// TwinCAT 3 PLC project Internship
// ProgramVersion: 3.1.4024.0
// libraries:
//   Tc2_Standard, * (Beckhoff Automation GmbH)
//   Tc2_System, * (Beckhoff Automation GmbH)
//   Tc3_Module, * (Beckhoff Automation GmbH)
// project tree:
//   Control/ FB_ControlSignal.TcPOU, FB_FeedForward.TcPOU, FB_PID.TcPOU, FB_Running.TcPOU (not stored), G_Mode.TcGVL
//   Filtering/ FB_Filtering.TcPOU, G_Filtered.TcGVL
//   GVL/ E_Mode.TcDUT, G_Enables.TcGVL, G_FilterConstants.TcGVL, G_OPC.TcGVL, G_Parameter.TcGVL
//   Inputs/Function Blocks/ FB_JoystickInputScaling.TcPOU, FB_Normalize.TcPOU, FB_Normalize_Joystick.TcPOU, FB_PositionInputScaling.TcPOU
//   Inputs/ G_Inputs.TcGVL
//   MotionRef/ FB_AutoClock.TcPOU, FB_DeadbandTester.TcPOU, FB_InitialPos.TcPOU, FB_MotionRef.TcPOU, FB_RunClock.TcPOU
//   Outputs/ FB_ValveOutput.TcPOU, G_Output.TcGVL
//   / PlcTask.TcTTO
//   Programs/ MAIN.TcPOU, P_ControlBlock.TcPOU, P_FeedForward.TcPOU, P_Filtering.TcPOU, P_Inputs.TcPOU, P_Modes.TcPOU, P_Output.TcPOU, P_PID.TcPOU, P_RunClock.TcPOU
//   XML/ FB_Derivator.TcPOU, G_Init.TcGVL, FB_Integrator.TcPOU
// real-time tasks:
//   TASK PlcTask: cycle T#1ms, priority 20, ADS port 350
// I/O:
//   DEVICE Device 3 (EtherCAT), AmsNetId 192.168.1.1.4.1
//     RIO (EK1100) [EK1100 EtherCAT Coupler (2A E-Bus)]
//       DI (EL1008) [EL1008 8Ch. Dig. Input 24V, 3ms]
//       DO (EL2008) [EL2008 8Ch. Dig. Output 24V, 0.5A]
//       AI1 (EL3068) [EL3068 8Ch. Ana. Input 0-10V]
//       AI2 (EL3068) [EL3068 8Ch. Ana. Input 0-10V]
//       AI3 (EL3174) [EL3174 4Ch. Ana. Input +/-10V Diff., +/-20mA SingleEnded, 16 Bit]
//       AO (EL4104) [EL4104 4Ch. Ana. Output 0-10V, 16bit]
//       End Cap (EL9011) [EL9011 End Terminal]
// variable links:
//   Internship/Internship Instance <-> Device 3 (EtherCAT)/RIO (EK1100)/AI1 (EL3068)
//     PlcTask Inputs/G_Inputs.nRawJoystick <-> AI Standard Channel 2/Value
//     PlcTask Inputs/G_Inputs.nRawPistonPosition <-> AI Standard Channel 3/Value
//   Internship/Internship Instance <-> Device 3 (EtherCAT)/RIO (EK1100)/AI2 (EL3068)
//     PlcTask Inputs/G_Inputs.nRawPa <-> AI Standard Channel 4/Value
//     PlcTask Inputs/G_Inputs.nRawPaLower <-> AI Standard Channel 5/Value
//     PlcTask Inputs/G_Inputs.nRawPb <-> AI Standard Channel 6/Value
//     PlcTask Inputs/G_Inputs.nRawPs <-> AI Standard Channel 1/Value
//   Internship/Internship Instance <-> Device 3 (EtherCAT)/RIO (EK1100)/AO (EL4104)
//     PlcTask Outputs/G_Output.nValveOutput <-> AO Output Channel 1/Analog output
//   Internship/Internship Instance <-> Device 3 (EtherCAT)/RIO (EK1100)/DI (EL1008)
//     PlcTask Inputs/G_Inputs.bAuto <-> Channel 1/Input
//     PlcTask Inputs/G_Inputs.bManual <-> Channel 2/Input
//     PlcTask Inputs/G_Inputs.bStartButton <-> Channel 3/Input
//     PlcTask Inputs/G_Inputs.bStopButton <-> Channel 4/Input
//   Internship/Internship Instance <-> Device 3 (EtherCAT)/RIO (EK1100)/DO (EL2008)
//     PlcTask Outputs/G_Output.bGreenLight <-> Channel 1/Output
//     PlcTask Outputs/G_Output.bRedLight <-> Channel 2/Output
//     PlcTask Outputs/G_Output.bRunning <-> Channel 3/Output

CONFIGURATION Internship
    RESOURCE PLC ON TwinCAT3
        TASK PlcTask(INTERVAL := T#1ms, PRIORITY := 20);
        PROGRAM MAIN WITH PlcTask : MAIN;
    END_RESOURCE
END_CONFIGURATION

// ---- GVL/E_Mode.TcDUT
{attribute 'qualified_only'}
{attribute 'strict'}
TYPE E_Mode :
(
	Off := 0,
	Auto := 1,
	Manuel := 2
);
END_TYPE

// ---- Control/G_Mode.TcGVL
{attribute 'qualified_only'}
VAR_GLOBAL
	bRunning : BOOL;
	bManual : BOOL;
	bAuto : BOOL;
END_VAR

// ---- Filtering/G_Filtered.TcGVL
{attribute 'qualified_only'}
VAR_GLOBAL
	fPressureSupplyFiltered		: LREAL;
	fPressurePistonSideFiltered : LREAL;
	fPressureRodSideFiltered 	: LREAL;
	fValveOutputFiltered		: LREAL;
	fValveOutputUnfiltered		: LREAL;
END_VAR

// ---- GVL/G_Enables.TcGVL
{attribute 'qualified_only'}
VAR_GLOBAL
	// Enables
	bEnablePID 		: BOOL := FALSE; // Enable PID Control
	bEnableU 		: BOOL := FALSE; // Enable Signal to Valve
	bEnableFF 		: BOOL := FALSE; // Enable FeedForward
	bMotionSelect 	: BOOL := FALSE; // Switch Motion Reference generator
	bEnableComp 	: BOOL := FALSE; // Driving with Compensator
	bDeadBand 		: BOOL := FALSE; // Enable Dead Band Testing
END_VAR

// ---- GVL/G_FilterConstants.TcGVL
{attribute 'qualified_only'}
VAR_GLOBAL
	// Filter constants
	fPressureFilterNum :LREAL := 0.003137;
	fPressureFilterDenz : LREAL := 1.0;
	fPressureFilterDen : LREAL := -0.9969;
	fPressureFilterInit : LREAL := 0.0;
	
	fSignalFilterNum : LREAL := 0.09516;
	fSignalFilterDenz : LREAL := 1.0;
	fSignalFilterDen : LREAL := -0.9048;
	fSignalFilterInit : LREAL := 0.0;
	
	fDerivatorFilterNum : LREAL := 0.0009995;
	fDerivatorFilterDenz : LREAL := 1.0;
	fDerivatorFilterDen : LREAL := -0.999;
	fDerivatorFilterInit : LREAL := 0.0;	
END_VAR

// ---- GVL/G_OPC.TcGVL
{attribute 'qualified_only'}
VAR_GLOBAL
	
	// Unfiltered Pressures
	fPa : LREAL;
	fPb : LREAL;
	fPs : LREAL;
	fPaLower : LREAL;
	
	// Filtered Pressures
	fPaFiltered : LREAL;
	fPbFiltered : LREAL;
	fPsFiltered : LREAL;
	fPaLowerFiltered : LREAL;
	
	
	fPistonPosition : LREAL;
	fJoystick : LREAL;
	
	fXRef : LREAL;
	fXDotRef : LREAL;
	
	fU : LREAL;
	fTime : LREAL;
	fError : LREAL;
	fSignalPID : LREAL;
	fUFF : LREAL;
END_VAR

// ---- GVL/G_Parameter.TcGVL
{attribute 'qualified_only'}
VAR_GLOBAL
	// Motion Ref
	fAmplitude : LREAL := 0.1;
	fMean : LREAL := 0.2;
	fFrequency : LREAL := 0.05;
	
	
	// Valve Values
	fQMaxDown : LREAL := 15.9;
	fQMaxUp : LREAL := 24.4;
	fDeadUp : LREAL := 0.13;
	fDeadDown : LREAL := 0.13;
	
	fMaxSpeed : LREAL := 0.01; // [m/s] 
	
	// Deadband test
	fConst : LREAL := 0.0; // [-1, 1]

	
	fCycleTime : LREAL := 0.001; // Time Step [s]
	fQConst : LREAL := 15;
	
	// PID-constants
	Kp : LREAL := 14.0; 	// P
	Ki : LREAL := 0.0;		// I
	Kd : LREAL := 0.0;		// D
	
	
	
	
END_VAR

// ---- Inputs/G_Inputs.TcGVL
{attribute 'qualified_only'}
VAR_GLOBAL
	// Mode Selector
	bManual 			AT %I* : BOOL;
	bAuto	 			AT %I* : BOOL;
	bStartButton		AT %I* : BOOL;
	bStopButton			AT %I* : BOOL;
	
	// Raw Pressure Values
	nRawPa 				AT %I*	: INT;
	nRawPb				AT %I*	: INT;
	nRawPs				AT %I*	: INT;
	nRawPaLower				AT %I* 	: INT;
	
	// Raw Position Values
	nRawPistonPosition 	AT %I*	: INT;
	nRawJoystick		AT %I*	: INT;
END_VAR

// ---- Outputs/G_Output.TcGVL
{attribute 'qualified_only'}
VAR_GLOBAL
	// Digital Outputs
	bGreenLight 			AT %Q* : BOOL;
	bRedLight 				AT %Q* : BOOL;
	
	// Analog Outputs
	nValveOutput 			AT %Q* : INT; 
	bRunning				AT %Q* : BOOL;
END_VAR

// ---- XML/G_Init.TcGVL
VAR_GLOBAL CONSTANT
	SS_INITIALIZE: SINT := 0;
	SS_STEP: SINT := 1;
END_VAR

// ---- Programs/MAIN.TcPOU
PROGRAM MAIN
VAR
END_VAR

P_Inputs();
P_Filtering();
P_ControlBlock();
P_Output();
//P_RunClock();
P_Modes();
P_PID();
P_FeedForward();

END_PROGRAM

// ---- Programs/P_Inputs.TcPOU
PROGRAM P_Inputs
VAR
	fbNormPa :  FB_Normalize;
	fbNormPb :  FB_Normalize;
	fbNormPs :  FB_Normalize;
	
	fbNormPistonPosition : FB_PositionInputScaling;
	fbJoystick : FB_JoystickInputScaling;

	fPa : LREAL;
	fPb : LREAL;
	fPs : LREAL;
	
	fPistonPosition : LREAL;
END_VAR

fbNormPa(
	nRawInput := G_Inputs.nRawPa,
	fMaxValue := 400.0, 			// [Bar]
	fNormalizedInput => G_OPC.fPa
);

fbNormPb(
	nRawInput := G_Inputs.nRawPb,
	fMaxValue := 400.0, 			// [Bar]
	fNormalizedInput => G_OPC.fPb
);

fbNormPs(
	nRawInput := G_Inputs.nRawPs,
	fMaxValue := 400.0, 			// [Bar]
	fNormalizedInput => G_OPC.fPs
);

fbNormPistonPosition(
	nRawInput := G_Inputs.nRawPistonPosition,
	fOutput => G_OPC.fPistonPosition
);
	
fbJoystick(
	nRawInput := G_Inputs.nRawJoystick,
	bEnable := G_Inputs.bManual,
	fOutput => G_OPC.fJoystick
);

END_PROGRAM

// ---- Inputs/Function Blocks/FB_Normalize.TcPOU
FUNCTION_BLOCK FB_Normalize
VAR_INPUT
	nRawInput : INT;
	fMaxValue : LREAL;
END_VAR
VAR_OUTPUT
	fNormalizedInput : LREAL;
END_VAR
VAR
END_VAR

fNormalizedInput := (fMaxValue	* INT_TO_LREAL(nRawInput)) / 32767.0;

fNormalizedInput := LIMIT(0, fNormalizedInput, fMaxValue);

END_FUNCTION_BLOCK

// ---- Inputs/Function Blocks/FB_PositionInputScaling.TcPOU
FUNCTION_BLOCK FB_PositionInputScaling
VAR_INPUT
	nRawInput : INT;
END_VAR
VAR_OUTPUT
	fOutput : LREAL;
END_VAR
VAR
	fRawInput : LREAL;
	fNormalizedInput: LREAL;
	fMaxInputValue 			: LREAL := 16099.0;
	fMinInputValue			: LREAL := 125.0;
	fMaxOutputValue  		: LREAL := 0.5;
	fMinOutputValue  		: LREAL := 0.0;		
END_VAR

fRawInput := INT_TO_LREAL(nRawInput);

fNormalizedInput := (fRawInput - fMinInputValue) / (fMaxInputValue - fMinInputValue);

fOutput := LIMIT(fMinOutputValue, fMinOutputValue + fNormalizedInput*(fMaxOutputValue - fMinOutputValue), fMaxOutputValue);

END_FUNCTION_BLOCK

// ---- Inputs/Function Blocks/FB_JoystickInputScaling.TcPOU
FUNCTION_BLOCK FB_JoystickInputScaling
VAR_INPUT
	bEnable : BOOL;
	nRawInput : INT;
END_VAR
VAR_OUTPUT
	fOutput : LREAL;
END_VAR
VAR
	fRawInput : LREAL;
	fTempInput : LREAL;
	fTempOutput : LREAL;
	fMaxInputValue			: LREAL := 14746.0;
	fMinInputValue 			: LREAL := 1617.0;
	fNeutralInputValue  	: LREAL := 8160.0;
	fNeutralDeadband		: LREAL := 100.0;
	fMaxOutputValue  		: LREAL := 1.0;
	fMinOutputValue  		: LREAL := -1.0;
	fNeutralOutputValue  	: LREAL := 0.0;
END_VAR

fRawInput := INT_TO_LREAL(nRawInput);

fTempInput := fRawInput - fNeutralInputValue;

IF fTempInput > fNeutralDeadband THEN
	fTempOutput := fTempInput/(fMaxInputValue - fNeutralInputValue);
ELSIF fTempInput < -fNeutralDeadband THEN	
	fTempOutput := fTempInput/(fNeutralInputValue - fMinInputValue);
ELSE
	fTempOutput := 0.0;
END_IF

IF NOT(bEnable) THEN
	fOutput := 0.0;
ELSE
	fOutput := LIMIT(fMinOutputValue, fTempOutput, fMaxOutputValue);
END_IF

END_FUNCTION_BLOCK

// ---- Programs/P_Filtering.TcPOU
PROGRAM P_Filtering
VAR
	//fbControlBlock : c_FB_ControlBlockWithMonito;
	fbFilterPa : FB_Filtering;
	fbFilterPb : FB_Filtering;
	fbFilterPs : FB_Filtering;
	fbFilterU : FB_Filtering;
	fbFilterPaLower : FB_Filtering;
END_VAR

fbFilterPa(
	ssMethodType := 1,
	Signal := G_OPC.fPa,
	Num := G_FilterConstants.fPressureFilterNum,
	Denz := G_FilterConstants.fPressureFilterDenz,
	Den := G_FilterConstants.fPressureFilterDen,
	Initial := G_FilterConstants.fPressureFilterInit,
	
	Signal_Filtered => G_Filtered.fPressurePistonSideFiltered,
	Signal_Filtered => G_OPC.fPaFiltered
);

fbFilterPb(
	ssMethodType := 1,
	Signal := G_OPC.fPb,
	Num := G_FilterConstants.fPressureFilterNum,
	Denz := G_FilterConstants.fPressureFilterDenz,
	Den := G_FilterConstants.fPressureFilterDen,
	Initial := G_FilterConstants.fPressureFilterInit,
	
	Signal_Filtered => G_Filtered.fPressureRodSideFiltered,
	Signal_Filtered => G_OPC.fPbFiltered
);

fbFilterPs(
	ssMethodType := 1,
	Signal := G_OPC.fPs,
	Num := G_FilterConstants.fPressureFilterNum,
	Denz := G_FilterConstants.fPressureFilterDenz,
	Den := G_FilterConstants.fPressureFilterDen,
	Initial := G_FilterConstants.fPressureFilterInit,
	
	Signal_Filtered => G_Filtered.fPressureSupplyFiltered,
	Signal_Filtered => G_OPC.fPsFiltered
);

fbFilterPaLower(
	ssMethodType := 1,
	Signal := G_OPC.fPaLower,
	Num := G_FilterConstants.fPressureFilterNum,
	Denz := G_FilterConstants.fPressureFilterDenz,
	Den := G_FilterConstants.fPressureFilterDen,
	Initial := G_FilterConstants.fPressureFilterInit,
	
	Signal_Filtered => G_Filtered.fPressureSupplyFiltered,
	Signal_Filtered => G_OPC.fPaLowerFiltered
);

//fbFilterU(
//	ssMethodType := 1,
//	Signal := G_Filtered.fValveOutputUnfiltered,
//	Num := G_FilterConstants.fSignalFilterNum,
//	Denz := G_FilterConstants.fSignalFilterDenz,
//	Den := G_FilterConstants.fSignalFilterDen,
//	Initial := G_FilterConstants.fSignalFilterInit,
//	
//	Signal_Filtered => G_Filtered.fValveOutputFiltered,
//	Signal_Filtered => G_OPC_UA.fFilteredSignal
//);

END_PROGRAM

// ---- Filtering/FB_Filtering.TcPOU
FUNCTION_BLOCK FB_Filtering
VAR_INPUT
	ssMethodType: SINT;
	Signal: LREAL;
	Num: LREAL;
	DenZ: LREAL;
	Den: LREAL;
	Initial: LREAL;
END_VAR
VAR_OUTPUT
	Signal_Unfiltered: LREAL;
	Signal_Filtered: LREAL;
END_VAR
VAR
	DiscreteTransferFcn1_icLoad: USINT;
	DiscreteTransferFcn1_states: LREAL;
	c_TmpSignalConversionAtDisc: ARRAY[0..1] OF LREAL;
END_VAR



CASE ssMethodType OF
    SS_INITIALIZE: 
        (* SystemInitialize for Atomic SubSystem: '<Root>/FB_Filtering' *)
        (* InitializeConditions for DiscreteTransferFcn: '<S1>/Discrete Transfer Fcn1' *)
        DiscreteTransferFcn1_icLoad := 1;
        (* End of SystemInitialize for SubSystem: '<Root>/FB_Filtering' *)
    SS_STEP: 
        (* Outputs for Atomic SubSystem: '<Root>/FB_Filtering' *)
        (* SignalConversion: '<S1>/TmpSignal ConversionAtDiscrete Transfer Fcn1Inport3' *)
        c_TmpSignalConversionAtDisc[0] := DenZ;
        c_TmpSignalConversionAtDisc[1] := Den;
        (* DiscreteTransferFcn: '<S1>/Discrete Transfer Fcn1' *)

        IF DiscreteTransferFcn1_icLoad <> 0 THEN 
            DiscreteTransferFcn1_states := Initial;
        END_IF;

        Signal_Filtered := Num * DiscreteTransferFcn1_states;
        (* End of DiscreteTransferFcn: '<S1>/Discrete Transfer Fcn1' *)
        

        (* SignalConversion: '<S1>/Signal' incorporates:
         *  Outport: '<Root>/Signal_Unfiltered' *)
        Signal_Unfiltered := Signal;
        (* Update for DiscreteTransferFcn: '<S1>/Discrete Transfer Fcn1' incorporates:
         *  SignalConversion: '<S1>/Signal' *)
        DiscreteTransferFcn1_icLoad := 0;
        DiscreteTransferFcn1_states := Signal - (c_TmpSignalConversionAtDisc[1] * DiscreteTransferFcn1_states);
        (* End of Outputs for SubSystem: '<Root>/FB_Filtering' *)
END_CASE;

END_FUNCTION_BLOCK

// ---- Programs/P_ControlBlock.TcPOU
PROGRAM P_ControlBlock
VAR
	fbDeadBandTester : FB_DeadbandTester;
	fbAutoClock : FB_AutoClock;
	fbMotionRef : FB_MotionRef;
	fbControl : FB_ControlSignal;
	fbInitialPos : FB_InitialPos;
END_VAR


fbControl(
	bEnableU := G_Enables.bEnableU,
	fQMaxUp := G_Parameter.fQMaxUp,
	fQMaxDown := G_Parameter.fQMaxDown,
	fDeadUp := G_Parameter.fDeadUp,
	fDeadDown := G_Parameter.fDeadDown,
);


IF G_Mode.bAuto AND G_Mode.bRunning THEN

fbInitialPos(
	bEnable := G_Inputs.bStartButton,
	fCurrentPos := G_OPC.fPistonPosition
);

fbAutoClock(
	fStart := G_Inputs.bStartButton,
	fRunning := G_Mode.bRunning,
	fCycle := G_Parameter.fCycleTime
);

fbMotionRef(
	fTime := fbAutoClock.fTime,
	fAmplitude := G_Parameter.fAmplitude,
	fInitialPos := fbInitialPos.fInitialPos,
	fFrequency := G_Parameter.fFrequency,
	fXDotRef => G_OPC.fXDotRef,
	fXRef => G_OPC.fXRef 
);

fbControl(
	fUFF := G_OPC.fUFF,
	fPID := G_OPC.fSignalPID,
	
	fU => G_OPC.fU
);

ELSIF G_Mode.bManual AND G_Mode.bRunning THEN

fbInitialPos(
	bEnable := G_Inputs.bStartButton,
	fCurrentPos := G_OPC.fPistonPosition
);

fbDeadBandTester(
	fInput := G_OPC.fJoystick,
	bEnable := G_Enables.bDeadBandTest,
	fConst := G_Parameter.fConst,
	fOutput => G_OPC.fU
);

//fbControl(
//	fUFF := G_OPC.fJoystick * G_Parameter.fMaxSpeed,
//	fPID := G_OPC.fSignalPID,
	
//	fU => G_OPC.fU
//);


END_IF

END_PROGRAM

// ---- MotionRef/FB_DeadbandTester.TcPOU
FUNCTION_BLOCK FB_DeadbandTester
VAR_INPUT
	fInput : LREAL;
	bEnable : BOOL;
	fConst : LREAL;
END_VAR
VAR_OUTPUT
	fOutput : LREAL;
END_VAR
VAR
	
END_VAR

IF bEnable THEN
	fOutput := fInput;
ELSE
	fOutput := fConst;
END_IF

END_FUNCTION_BLOCK

// ---- MotionRef/FB_AutoClock.TcPOU
FUNCTION_BLOCK FB_AutoClock
VAR_INPUT
	fStart : BOOL;
	fRunning : BOOL;
	fCycle : LREAL;
END_VAR
VAR_OUTPUT
	fTime : LREAL;
END_VAR
VAR
END_VAR


IF NOT(fStart) OR NOT(fRunning) THEN
	fTime := 0.0;
ELSIF fStart AND fRunning THEN
	fTime := fTime + fCycle;		
END_IF

END_FUNCTION_BLOCK

// ---- MotionRef/FB_MotionRef.TcPOU
FUNCTION_BLOCK FB_MotionRef
VAR_INPUT
	fTime : LREAL;
	fAmplitude : LREAL;
	fFrequency : LREAL;
	fInitialPos : LREAL;
END_VAR
VAR_OUTPUT
	fXDotRef : LREAL;
	fXRef : LREAL;
END_VAR
VAR
	fPI : LREAL := 3.1415;
	fMean : LREAL;
END_VAR

fMean := fAmplitude + fInitialPos; 
fXRef := fMean - fAmplitude * COS(2*fPI * fFrequency * fTime);
fXDotRef := 2 * fPI *fFrequency * fAmplitude * SIN(2*fPI * fFrequency * fTime);

END_FUNCTION_BLOCK

// ---- Control/FB_ControlSignal.TcPOU
FUNCTION_BLOCK FB_ControlSignal
VAR_INPUT
	fUFF : LREAL;
	fPID : LREAL;
	bEnableU : BOOL;
	fQMaxUp 	: LREAL; // Needs to be positive (22)
	fQMaxDown 	: LREAL; // Needs to be positive (15)
	fDeadUp		: LREAL; // Needs to be positive (0.155)
	fDeadDown 	: LREAL; // Needs to be positive (0.18)
END_VAR
VAR_OUTPUT
	fU : LREAL;
END_VAR
VAR

	fUTemp : LREAL;
	fUTemp2 : LREAL;
	fUMax : LREAL := 0.9;
END_VAR

IF bEnableU THEN
	fUTemp := fUFF - fPID;
	
	// Deadband compensation
	IF fUTemp < 0.0 THEN	// Upwards
		fUTemp2 := fUTemp - fDeadUp;
	ELSIF fUTemp > 0.0 THEN // Downwards
		fUTemp2 := fUTemp + fDeadDown;
	ELSE
		fUTemp2 := 0.0;
	END_IF
	
	
	IF fUFF = 0 THEN
		fU := 0.0;
	ELSIF fUTemp2 >= fUMax THEN
		fU := fUMax;
	ELSIF fUTemp2 <= -fUMax THEN
		fU := -fUMax;
	ELSE
		fU := fUTemp2;
	END_IF
END_IF

END_FUNCTION_BLOCK

// ---- MotionRef/FB_InitialPos.TcPOU
FUNCTION_BLOCK FB_InitialPos
VAR_INPUT
	bEnable : BOOL;
	fCurrentPos : LREAL;
END_VAR
VAR_OUTPUT
	fInitialPos : LREAL;
END_VAR
VAR
END_VAR

IF bEnable THEN
	fInitialPos := fInitialPos;
ELSE 
	fInitialPos := fCurrentPos;
END_IF

END_FUNCTION_BLOCK

// ---- Programs/P_Output.TcPOU
PROGRAM P_Output
VAR
	fbValveOutput : FB_ValveOutput;
END_VAR

fbValveOutput(
	fNormalizedInput := G_OPC.fU,
	bEnable := G_Enables.bEnableU,
	nOutput => G_Output.nValveOutput	
);

IF G_Mode.bRunning THEN
	G_Output.bGreenLight := TRUE;
	G_Output.bRedLight := TRUE;
ELSE
	G_Output.bGreenLight := FALSE;
	G_Output.bRedLight := FALSE;
END_IF

END_PROGRAM

// ---- Outputs/FB_ValveOutput.TcPOU
FUNCTION_BLOCK FB_ValveOutput
VAR_INPUT
	bEnable 			: BOOL;
	fNormalizedInput 	: LREAL;
END_VAR
VAR_OUTPUT
	nOutput : INT; 
END_VAR
VAR
	nOffset 	: LREAL := 19630.0;
	nMaxValue	: LREAL := 29460.0;
	nMinValue 	: LREAL :=  9830.0;
	nTempOutput : LREAL;
END_VAR


IF fNormalizedInput > 0.0 THEN
	nTempOutput := (fNormalizedInput) * (nMaxValue - nOffset) + nOffset;
ELSIF fNormalizedInput < 0.0 THEN
	nTempOutput := (fNormalizedInput) * (nOffset - nMinValue) + nOffset;
ELSE 
	nTempOutput := nOffset;
END_IF



IF NOT(bEnable) THEN
	nOutput := LREAL_TO_INT(nOffset);
ELSIF (bEnable) THEN
	nOutput := LREAL_TO_INT(nTempOutput);	
END_IF

END_FUNCTION_BLOCK

// ---- Programs/P_Modes.TcPOU
PROGRAM P_Modes
VAR
	fbRunning : FB_Running;
END_VAR

fbRunning(
	bAuto := G_Inputs.bAuto,
	bManual := G_Inputs.bManual,
	bStart := G_Inputs.bStartButton,
	bStop := G_Inputs.bStopButton,
	
	bRunning => G_Mode.bRunning,
	bRunning => G_Output.bRunning,
	bManualMode => G_Mode.bManual,
	bAutoMode => G_Mode.bAuto
);

END_PROGRAM

// ---- Programs/P_PID.TcPOU
PROGRAM P_PID
VAR
	fbPID : FB_PID;
	fbIntegrator : FB_Integrator;
	fbDerivator : FB_Derivator;
	fbDerivatorFiltering : FB_Filtering;
END_VAR

IF (G_Enables.bEnablePID) THEN
	
	fbderivatorFiltering(
		ssMethodType := 1,
		Signal := fbPID.fSignalD,
		Num := G_FilterConstants.fDerivatorFilterNum,
		Denz := G_FilterConstants.fDerivatorFilterDenz,
		Den := G_FilterConstants.fDerivatorFilterDen,
		Initial := G_FilterConstants.fDerivatorFilterInit,
		Signal_Filtered => fbDerivator.fSignal
	);

	fbPID(
		fX := G_OPC.fXRef,
		fXReal := G_OPC.fPistonPosition,
		fKp := G_Parameter.Kp,
		fKi := G_Parameter.Ki,
		fKd := G_Parameter.Kd,
		
		fSignalI => fbIntegrator.fSignal,
		fSignalD => fbDerivatorFiltering.Signal_Filtered,
		
		fSignalIntegrated := fbIntegrator.fSignalIntegrated,
		fSignalDerivated := fbDerivator.fSignalDerivative,
		
		fError => G_OPC.fError,
		fSignalAdjusted => G_OPC.fSignalPID
	);

END_IF

END_PROGRAM

// ---- Control/FB_PID.TcPOU
FUNCTION_BLOCK FB_PID
VAR_INPUT
	fX : LREAL;
	fXReal : LREAL;
	fSignalIntegrated : LREAL;
	fSignalDerivated : LREAL;
	fKp : LREAL;
	fKi : LREAL;
	fKd : LREAL;
END_VAR
VAR_OUTPUT
	fSignalI : LREAL;
	fSignalD : LREAL;
	fSignalAdjusted : LREAL;
	fError  : LREAL;
END_VAR
VAR
	fTempP : LREAL;
	fTempI : LREAL;
	fTempD : LREAL;
	fTempOut : LREAL;
END_VAR

fError := fX - fXReal;

fSignalI := fError;
fSignalD := fError;

fTempP := fError * fKp;
fTempI := fSignalIntegrated * fKi;
fTempD := fSignalDerivated * fKd;

fTempOut := fTempP + fTempI + fTempD;

IF fTempOut > 1.0 THEN
	fSignalAdjusted := 1.0;
ELSIF fTempOut < -1.0 THEN
	fSignalAdjusted := -1.0;
ELSE
	fSignalAdjusted := fTempOut;
END_IF

END_FUNCTION_BLOCK

// ---- XML/FB_Integrator.TcPOU
FUNCTION_BLOCK FB_Integrator
VAR_INPUT
	ssMethodType: SINT;
	fSignal: LREAL;
END_VAR
VAR_OUTPUT
	fSignalIntegrated: LREAL;
END_VAR
VAR
	c_DiscreteTimeIntegrator_DS: LREAL;
END_VAR



CASE ssMethodType OF
    SS_INITIALIZE: 
        (* SystemInitialize for Atomic SubSystem: '<Root>/Integrator' *)
        (* InitializeConditions for DiscreteIntegrator: '<S1>/Discrete-Time Integrator' *)
        c_DiscreteTimeIntegrator_DS := 0.0;
        (* End of SystemInitialize for SubSystem: '<Root>/Integrator' *)
    SS_STEP: 
        (* Outputs for Atomic SubSystem: '<Root>/Integrator' *)
        (* Outport: '<Root>/fSignalIntegrated' incorporates:
         *  DiscreteIntegrator: '<S1>/Discrete-Time Integrator' *)
        fSignalIntegrated := c_DiscreteTimeIntegrator_DS;
        (* Update for DiscreteIntegrator: '<S1>/Discrete-Time Integrator' *)
        c_DiscreteTimeIntegrator_DS := (0.001 * fSignal) + c_DiscreteTimeIntegrator_DS;
        (* End of Outputs for SubSystem: '<Root>/Integrator' *)
END_CASE;

END_FUNCTION_BLOCK

// ---- XML/FB_Derivator.TcPOU
FUNCTION_BLOCK FB_Derivator
VAR_INPUT
	ssMethodType: SINT;
	fSignal: LREAL;
END_VAR
VAR_OUTPUT
	fSignalDerivative: LREAL;
END_VAR
VAR
	rtb_TSamp: LREAL;
	UD_DSTATE: LREAL;
END_VAR



CASE ssMethodType OF
    SS_INITIALIZE: 
        (* SystemInitialize for Atomic SubSystem: '<Root>/Derivator' *)
        (* InitializeConditions for UnitDelay: '<S2>/UD'
         *
         * Block description for '<S2>/UD':
         *  
         *  Store in Global RAM *)
        UD_DSTATE := 0.0;
        (* End of SystemInitialize for SubSystem: '<Root>/Derivator' *)
    SS_STEP: 
        (* Outputs for Atomic SubSystem: '<Root>/Derivator' *)
        (* SampleTimeMath: '<S2>/TSamp'
         *
         * About '<S2>/TSamp':
         *  y = u * K where K = 1 / ( w * Ts )
         *   *)
        rtb_TSamp := fSignal * 1000.0;
        (* Outport: '<Root>/fSignalDerivative' incorporates:
         *  Sum: '<S2>/Diff'
         *  UnitDelay: '<S2>/UD'
         *
         * Block description for '<S2>/Diff':
         *  
         *  Add in CPU
         *
         * Block description for '<S2>/UD':
         *  
         *  Store in Global RAM *)
        fSignalDerivative := rtb_TSamp - UD_DSTATE;
        (* Update for UnitDelay: '<S2>/UD'
         *
         * Block description for '<S2>/UD':
         *  
         *  Store in Global RAM *)
        UD_DSTATE := rtb_TSamp;
        (* End of Outputs for SubSystem: '<Root>/Derivator' *)
END_CASE;

END_FUNCTION_BLOCK

// ---- Programs/P_FeedForward.TcPOU
PROGRAM P_FeedForward
VAR
	fbFF : FB_FeedForward;
END_VAR

IF (G_Enables.bEnableFF AND G_Mode.bRunning) THEN
fbFF(
	fXDotRef := G_OPC.fXDotRef,
	fQMaxUp := G_Parameter.fQMaxUp,
	fQMaxDown := G_Parameter.fQMaxDown,
	fDeadUp := G_Parameter.fDeadUp,
	fDeadDown := G_Parameter.fDeadDown,
	
	fUFF => G_OPC.fUFF
);
END_IF

END_PROGRAM

// ---- Control/FB_FeedForward.TcPOU
FUNCTION_BLOCK FB_FeedForward
VAR_INPUT
	fXDotRef 	: LREAL; // Motion Referance
	fQMaxUp 	: LREAL; // Needs to be positive (22)
	fQMaxDown 	: LREAL; // Needs to be positive (15)
	fDeadUp		: LREAL; // Needs to be positive (0.155)
	fDeadDown 	: LREAL; // Needs to be positive (0.18)
END_VAR
VAR_OUTPUT
	fUFF : LREAL;
END_VAR
VAR
	fUTemp : LREAL;
	fUMax : LREAL := 0.9;
	fQRef : LREAL;
	fAp : LREAL := 33.1 / 10000.0;
	fAa : LREAL := 23.56 / 10000.0;
END_VAR


IF fXDotRef >= 0.0 THEN // Upwards
	
	fQRef := fAp * fXDotRef * 60000;
	fUTemp := -((fQRef/fQMaxUp) * (fUMax-fDeadUp));
	
//	IF fUTemp < -fUMax THEN
//		fUFF := -fUMax;
	
//	ELSIF fUTemp > -fDeadUp THEN
//		fUFF := -fDeadUp;
//	ELSE
//		fUFF := fUTemp;
//	END_IF

ELSIF fXDotRef < 0.0 THEN // Downwards
	
	fQRef := fAa * fXDotRef * 60000;
	fUTemp := -((fQRef/fQMaxDown) * (fUMax-fDeadDown)); // FDeadDown needs to be positive
	
//	IF fUTemp > fUMax THEN
//		fUFF := fUMax;
	
//	ELSIF fUTemp < fDeadDown THEN
//		fUFF := fDeadDown;
//	ELSE
//		fUFF := fUTemp;
//	END_IF

END_IF

fUFF := fUTemp; // Tomec

END_FUNCTION_BLOCK

// ---- Inputs/Function Blocks/FB_Normalize_Joystick.TcPOU
FUNCTION_BLOCK FB_Normalize_Joystick
VAR_INPUT
	nRawInput : INT;
END_VAR
VAR_OUTPUT
	fNormalizedInput : LREAL;
END_VAR
VAR
END_VAR

fNormalizedInput := (INT_TO_LREAL(nRawInput) - 32767.0/2.0) / (32767.0/2.0);

fNormalizedInput := LIMIT(-1, fNormalizedInput, 1);

END_FUNCTION_BLOCK

// ---- MotionRef/FB_RunClock.TcPOU
FUNCTION_BLOCK FB_RunClock
VAR_INPUT
	bStart 		: BOOL;
	bStop 		: BOOL;
	fCycleTime  : LREAL;
END_VAR
VAR_OUTPUT
	fTime : LREAL;
END_VAR
VAR
	bOnOff : BOOL;
END_VAR

IF bStop OR (G_Work.eStatus = E_Status.Off) THEN
	bOnOff := FALSE;
	fTime := 0.0;
ELSIF bOnOff OR bStart THEN
	bOnOff := TRUE;
	fTime := fTime + fCycleTime;
END_IF

END_FUNCTION_BLOCK

// ---- Programs/P_RunClock.TcPOU
PROGRAM P_RunClock
VAR
	fbRunClock : FB_RunClock;
END_VAR

fbRunClock(
	bStart := TRUE,
	bStop := G_Inputs.bStopButton,
	fCycleTime := G_Parameter.fCycleTime,
	
	fTime => G_OPC.fTime
);

END_PROGRAM
